FUNCTION_BLOCK RunUnitControllerV2 EXTENDS RunGroupNode
VAR_INPUT
	isEmergency : BOOL; //would trigger initialize , raise alarm
	isSafetyFault : BOOL;
	isAirIncorrect : BOOL;
	
	isManual : BOOL;
	
	requestInit : bool;
	requestErrorClear AT%M* : eErrorClearWays := eErrorClearWays.NO_ACTION;
	
	marshal : POINTER TO RunUnitGeneric;
END_VAR
VAR_OUTPUT
	//------------------------
	//	Error handling channel
	//------------------------	
	errorType AT%Q* : eCategrories;
	errorIndex AT%Q* : DINT;
	errorCode AT%Q* : UDINT;
	
END_VAR
VAR		
	//error
	errorDevice : POINTER TO CommonBase := 0; //null reference	
	errorDelayDetect : TON;	
	
	needInit : BOOL;
END_VAR
VAR PERSISTENT
	axisUpperBound : INT;
	cylinderUpperBound : INT;
	signalUpperBound : INT;
	unitUpperBound : INT;
	slotUpperBound : int;
END_VAR
VAR CONSTANT
	ERR_EMG : DWORD :=1;
	ERR_INCORRECT_AIR : DWORD :=10;
	ERR_SAFETY : DWORD :=8501;
END_VAR

//Purpose:
// 1. As abstract machine itself , switch between modes 
// 2. bridge signals to coordinator

//Clarify : 
// 1. Manual mode : component driven only
// 2. Semi-auto (PAUSE) : sequencer were driven, but most are forbidden to execute (PAUSE state)
// 3. Auto: sequencer drive , all drive autonomous

//Difference to V1 
//1. Hierarchy initializing

//----------------------
//	Components level
//----------------------
FOR nCounter :=1 TO axisUpperBound BY 1 DO
	gvl.axisControls[nCounter]();
END_FOR
FOR nCounter :=1 TO cylinderUpperBound BY 1 DO
	gvl.pnuematicControls[nCounter]^();
END_FOR
FOR nCounter :=1 TO signalUpperBound BY 1 DO
	gvl.signalControls[nCounter]();
END_FOR
//---------------------------
//	System LEVEL
//---------------------------
IF isEmergency AND errorDelayDetect.Q   THEN
	//Emergency pressed
	//errorDevice := marshal;
	marshal^.AlarmCode := ERR_EMG;
	errorIndex := 1;
	errorDevice := marshal;
ELSIF isSafetyFault AND errorDelayDetect.Q THEN
	//Safety
	//errorDevice := marshal;
	marshal^.AlarmCode := ERR_SAFETY;
	errorIndex := 1;
	errorDevice := marshal;
ELSIF isAirIncorrect AND errorDelayDetect.Q  THEN
	//Air supply
	//errorDevice := marshal;
	marshal^.AlarmCode := ERR_INCORRECT_AIR;
	errorIndex := 1;
	errorDevice := marshal;
ELSE
	//----------------------------------------
	// 	COMPONENT LEVEL:
	//	running all devices/detect errors
	//----------------------------------------
	FOR nCounter :=1 TO axisUpperBound BY 1 DO
		//error detection
		IF errorDevice=0 AND errorDelayDetect.Q AND gvl.axisControls[nCounter].ErrorDetect() <> 0 THEN
			//error scaned
			errorIndex := nCounter;
			errorDevice := ADR(gvl.axisControls[nCounter]);
		END_IF
	END_FOR
	FOR nCounter :=1 TO cylinderUpperBound BY 1 DO
		//error detection
		IF errorDevice=0 AND errorDelayDetect.Q AND gvl.pnuematicControls[nCounter]^.ErrorDetect() <> 0 THEN
			//error scaned
			errorIndex := nCounter;
			errorDevice := gvl.pnuematicControls[nCounter];
		END_IF
	END_FOR
	FOR nCounter :=1 TO unitUpperBound BY 1 DO
		//error detection
		IF errorDevice=0 AND errorDelayDetect.Q AND gvl.units[nCounter] <> 0 AND_THEN gvl.units[nCounter]^.ErrorDetect() <> 0THEN
			//station
			errorIndex := nCounter;
			errorDevice := gvl.units[nCounter];
		END_IF
	END_FOR
END_IF


//routines
errorDelayDetect(IN:= (errorDevice = 0), PT:= T#200MS, Q=> , ET=> );	//after reset , wait 100ms to detect
IF errorDevice <>0 THEN
	//error index had been specified
	errorType := errorDevice^.TypeCode();
	errorCode := errorDevice^.ErrorDetect();
	
	//reset error handling
	IF requestErrorClear <> eErrorClearWays.NO_ACTION THEN
		errorDevice^.ErrorClear(requestErrorClear); //call error clear function
		errorDevice := 0 ;// cut link
	END_IF
	
	
ELSE
	//reset
	errorType := 0;
	errorIndex := 0;
	errorCode := 0;
END_IF
AlarmCode := SHL(TO_UDINT(errorType),24) +  TO_UDINT(SHL(errorIndex,16)) + TO_UDINT(errorCode);

//-------------------------------------------------
// START/STOP (internal pause due to process error
//-------------------------------------------------
IF errorDevice <>0  THEN
	bPause := TRUE; //forced stop
ELSE
	//leave current status
END_IF
//------------------------------------------------------------
//	IN MANUAL MODE, FORBIDEEN TO DRIVE SEQUENCES
//------------------------------------------------------------
IF NOT isManual THEN
	// sequences driven
	FOR nCounter :=1 TO unitUpperBound BY 1 DO
		IF gvl.units[nCounter] <> 0 THEN
			gvl.units[nCounter]^();
		END_IF
	END_FOR
END_IF

//-------------------
//	Check whether init condition
//, TODO or fatal situation
//-------------------
IF NOT needInit AND isEmergency THEN
	needInit := TRUE;
END_IF

SUPER^(); //state machine driven
CASE outputState OF
	eSpecialStates.MAIN_WAIT_INITIALIZING:
		bSerialTransition := requestInit AND NOT isEmergency;
		IF bSerialTransition THEN
			needInit := FALSE; //reset
		END_IF
	eSpecialStates.MAIN_INITIALIZING:
		bSerialTransition := marshal<>0 AND_THEN marshal^.Initialize();
		IF bSerialTransition THEN
			marshal^.NextState := eSpecialStates.GENERIC_GROUP_START;
		END_IF
	eSpecialStates.MAIN_INITIALIZED:
		//wait emergency situation 
		IF needInit OR requestInit THEN
			NextState := eSpecialStates.MAIN_WAIT_INITIALIZING;
		END_IF
END_CASE

METHOD FB_init : BOOL
VAR_INPUT
	bInitRetains : BOOL; // if TRUE, the retain variables are initialized (warm start / cold start)
	bInCopyCode : BOOL;  // if TRUE, the instance afterwards gets moved into the copy code (online change)
	
	argParent : POINTER TO RunUnitGeneric;
	argSlotBase : POINTER TO RunMaterial;
	argSlotLast : POINTER TO RunMaterial;
	
END_VAR
//initialize 
Parent := argParent;
SlotBase := argSlotBase;
SlotLast := argSlotLast;
//
IF bInitRetains THEN
	NextState := eSpecialStates.INITIAL_BEGIN;
	
	// Semi-statically setup running index bound
	axisUpperBound := SIZEOF(gvl.axisControls)/SIZEOF(gvl.axisControls[1]);
	cylinderUpperBound := SIZEOF(gvl.cylinderControls)/SIZEOF(gvl.cylinderControls[1]);
	signalUpperBound := SIZEOF(gvl.signalControls)/SIZEOF(gvl.signalControls[1]);
	unitUpperBound := SIZEOF(gvl.units)/SIZEOF(gvl.units[1]);
	slotUpperBound := SIZEOF(gvl.materialSlots)/SIZEOF(gvl.materialSlots[1]);
	
END_IF

state := eSpecialStates.MAIN_INITIALIZING; //as beginning
NextState:=state;
END_METHOD

END_FUNCTION_BLOCK

(* stored: Version 1.1.0.1, ProductVersion 3.1.4024.0
   POU RunUnitControllerV2: Id {b8ed3dbb-ffb0-4792-8cf6-5dee6569b3ad}, SpecialFunc None
   Method FB_init: Id {59012378-cdc1-4f5d-9c82-ed2cdadc0d0a} *)
